TYPE ST_ErrorSection EXTENDS ST_SectionBase :
STRUCT
	nErrCount	: UINT;
	
	
END_STRUCT
END_TYPE

(* stored: Version 1.1.0.1, ProductVersion 3.1.4024.12
   DUT ST_ErrorSection: Id {3f9e29ab-89bd-4ef5-9165-a474bc131d81} *)
